Fanuc KAREL source: kt00745.KL

-- PROVISIONAL review KL for V1013-1; original PC SHA256 871bc67ab2824bc764b16f602010056297b79c61be11a502df18102220fd99b1
-- Incomplete behavior may be omitted. Consult companion uncertainty JSON. Do not deploy.
PROGRAM KT00745
%NOLOCKGROUP
BEGIN
  -- UNRESOLVED_PC offsets 5-18; opcodes 22,1D,23
  -- UNRESOLVED_PC offsets 23-27; opcodes 7F
END KT00745
